// TIA Portal V20 export
// export: Created 2025-12-01T14:57:21.8658901Z, ExportSetting None, DisplayName Totally Integrated Automation Portal, DisplayVersion V20 Update 3, DisplayName TIA Portal Openness, DisplayVersion V20 Update 3, DisplayName TIA Portal Version Control Interface, DisplayVersion V20 Update 3, DisplayName STEP 7 Professional, DisplayVersion V20 Update 3, DisplayName STEP 7 Safety, DisplayVersion V20 Update 2, DisplayName WinCC Basic/Comfort/Advanced, DisplayVersion V20 Update 3, DisplayName WinCC Professional, DisplayVersion V20 Update 3, DisplayName WinCC Unified, DisplayVersion V20 Update 3
FUNCTION "FC5_Tratar_Pantalla" : Void   // FC5, LAD
{ S7_Optimized_Access := 'FALSE' }
AUTHOR : PANTALLA
NAME : 20160413
VERSION : 3.3
// stored: AutoNumber false, SetENOAutomatically false
BEGIN

REGION Network 1: Que PLC es? CCPIF A o CCPIF B o CCPIF C
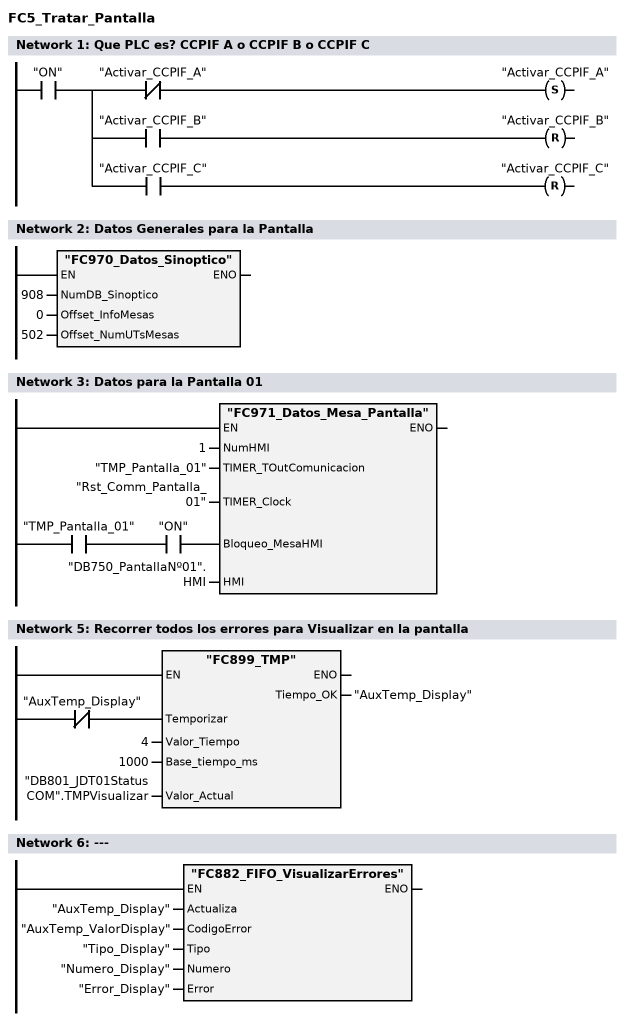
   RUNG wire#powerrail
      Contact( "ON" )
      wire#w1
      I_Contact( "Activar_CCPIF_A" )
      S_Coil( "Activar_CCPIF_A" )
   END_RUNG
   RUNG wire#w1
      Contact( "Activar_CCPIF_B" )
      R_Coil( "Activar_CCPIF_B" )
   END_RUNG
   RUNG wire#w1
      Contact( "Activar_CCPIF_C" )
      R_Coil( "Activar_CCPIF_C" )
   END_RUNG
   // the same network as SCL:
   IF "ON" AND NOT "Activar_CCPIF_A" THEN "Activar_CCPIF_A" := TRUE; END_IF;
   IF "ON" AND "Activar_CCPIF_B" THEN "Activar_CCPIF_B" := FALSE; END_IF;
   IF "ON" AND "Activar_CCPIF_C" THEN "Activar_CCPIF_C" := FALSE; END_IF;
END_REGION

REGION Network 2: Datos Generales para la Pantalla
   RUNG wire#powerrail
      "FC970_Datos_Sinoptico"(NumDB_Sinoptico := 908, Offset_InfoMesas := 0, Offset_NumUTsMesas := 502)
   END_RUNG
   // the same network as SCL:
   "FC970_Datos_Sinoptico"(NumDB_Sinoptico := 908, Offset_InfoMesas := 0, Offset_NumUTsMesas := 502);
END_REGION

REGION Network 3: Datos para la Pantalla 01
   RUNG wire#powerrail
      "FC971_Datos_Mesa_Pantalla"(Bloqueo_MesaHMI := wire#w1, NumHMI := 1, TIMER_TOutComunicacion := "TMP_Pantalla_01", TIMER_Clock := "Rst_Comm_Pantalla_01", HMI := "DB750_PantallaNº01".HMI)
   END_RUNG
   RUNG wire#powerrail
      Contact( "TMP_Pantalla_01" )
      Contact( "ON" )
   END_RUNG wire#w1
   // the same network as SCL:
   "FC971_Datos_Mesa_Pantalla"(NumHMI := 1,
                           TIMER_TOutComunicacion := "TMP_Pantalla_01",
                           TIMER_Clock := "Rst_Comm_Pantalla_01",
                           Bloqueo_MesaHMI := "TMP_Pantalla_01" AND "ON",
                           HMI := "DB750_PantallaNº01".HMI);
END_REGION

REGION Network 4: ANADIR TANTAS PANTALLAS COMO EXISTAN EN EL PROYECTO
END_REGION

REGION Network 5: Recorrer todos los errores para Visualizar en la pantalla
   RUNG wire#powerrail
      "FC899_TMP"(Valor_Tiempo := 4, Base_tiempo_ms := 1000, Tiempo_OK => "AuxTemp_Display", Valor_Actual := "DB801_JDT01StatusCOM".TMPVisualizar, Temporizar := wire#w1)
   END_RUNG
   RUNG wire#powerrail
      I_Contact( "AuxTemp_Display" )
   END_RUNG wire#w1
   // the same network as SCL:
   "FC899_TMP"(Temporizar := NOT "AuxTemp_Display",
               Valor_Tiempo := 4,
               Base_tiempo_ms := 1000,
               Valor_Actual := "DB801_JDT01StatusCOM".TMPVisualizar,
               Tiempo_OK => "AuxTemp_Display");
END_REGION

REGION Network 6: ---
   RUNG wire#powerrail
      "FC882_FIFO_VisualizarErrores"(Actualiza := "AuxTemp_Display", CodigoError := "AuxTemp_ValorDisplay", Tipo := "Tipo_Display", Numero := "Numero_Display", Error := "Error_Display")
   END_RUNG
   // the same network as SCL:
   "FC882_FIFO_VisualizarErrores"(Actualiza := "AuxTemp_Display",
                           CodigoError := "AuxTemp_ValorDisplay",
                           Tipo := "Tipo_Display",
                           Numero := "Numero_Display",
                           Error := "Error_Display");
END_REGION
END_FUNCTION
